FUNCTION_BLOCK FB_EL3152
VAR_INPUT PERSISTENT

	deviceConfig    : EL3152_DEV_CONFIG; // Configuration settings for the CT121F device
	
END_VAR
VAR_OUTPUT
		
	Channel1  : REAL;
	Channel2  : REAL;
	
END_VAR
VAR
	    PDOS : EL3052_PDOS; // Process Data Objects for RWPT01D communication
END_VAR


_AnalogInputs();

METHOD PRIVATE _AnalogInputs
VAR_INPUT
END_VAR
// Calculate the actual motor speed
Channel1 := _Scale(
    X := DINT_TO_REAL(PDOS.HwToPLC.Channel1.Value), 
    I_LO := deviceConfig.channel1InputLow, 
    I_HI := deviceConfig.channel1InputHigh, 
    O_LO := deviceConfig.channel1OutputLow, 
    O_HI := deviceConfig.channel1OutputHigh
);

// Calculate the actual motor speed
Channel2 := _Scale(
    X := DINT_TO_REAL(PDOS.HwToPLC.Channel2.Value), 
    I_LO := deviceConfig.channe12InputLow, 
    I_HI := deviceConfig.channe12InputHigh, 
    O_LO := deviceConfig.channe12OutputLow, 
    O_HI := deviceConfig.channe12OutputHigh
);
END_METHOD

METHOD PRIVATE _Scale : REAL
VAR_INPUT
	
	X : REAL;
	I_LO : REAL;
	I_HI : REAL;
	O_LO : REAL;
	O_HI : REAL;
	
END_VAR
IF I_LO = I_HI THEN
	_Scale := O_LO;
ELSE
	_Scale := (O_HI - O_LO) / (I_HI - I_LO) * (LIMIT(I_LO, X, I_HI) - I_LO) + O_LO;
END_IF;
END_METHOD

END_FUNCTION_BLOCK

(* stored: Version 1.1.0.1, ProductVersion 3.1.4024.15
   POU FB_EL3152: Id {45f1f3b5-f79d-4535-8823-23cd1a6657ba}, SpecialFunc None
   Method _AnalogInputs: Id {ecdb5f49-2bec-4ebb-a2da-f364805c28ef}
   Method _Scale: Id {2ac0f6b0-ef77-4731-9a36-6e4fb1e78a1f} *)
